{attribute 'GeneratedUsingTerminal: EJ7031-0000-0026'}
{attribute addProperty BoxType "EJ7031-0000-0026"}
{attribute addProperty Id "AdsAddrAT %I*.TcoAmsAddr0Chn0AT %I*USINT1Chn1AT %I*USINT1StateAT %I*UINT2"}
{attribute addProperty CRC "995053194"}
{attribute addProperty Size "4"}
TYPE InfoData_3B4F4E8A :
STRUCT
	{attribute addProperty Name "AdsAddr"}
	AdsAddr AT %I* : .TcoAmsAddr;
	{attribute addProperty Name "Chn0"}
	Chn0 AT %I* : USINT;
	{attribute addProperty Name "Chn1"}
	Chn1 AT %I* : USINT;
	{attribute addProperty Name "State"}
	State AT %I* : UINT;
END_STRUCT
END_TYPE

(* stored: Version 1.2.0.0, ProductVersion 3.1.4024.9
   DUT InfoData_3B4F4E8A: Id {5ba50729-1077-4e56-9cc1-18ef95fa5931} *)
